FUNCTION_BLOCK FB_Timeout
VAR_INPUT
	bActivate			: BOOL;
	tDuration			: TIME;
END_VAR
VAR_OUTPUT
	nAttempts			: USINT := 0;
END_VAR
VAR
	bTimerEnable		: BOOL := TRUE;
	tmrTimeoutTimer		: Tc2_Standard.TON;
END_VAR

IF bActivate THEN
	tmrTimeoutTimer(IN := bTimerEnable, PT := tDuration);
	IF tmrTimeoutTimer.Q THEN
		nAttempts := nAttempts + 1;
		tmrTimeoutTimer(IN := FALSE);
	END_IF
	
ELSE
	nAttempts := 0;
	bTimerEnable := TRUE;
END_IF

END_FUNCTION_BLOCK

(* stored: Version 1.1.0.1, ProductVersion 3.1.4024.11
   POU FB_Timeout: Id {8b3cd484-6b5d-4ac8-952c-5394659be4cb}, SpecialFunc None *)
